// SIMATIC S7-200 project (STEP 7-Micro/WIN), CPU 224 REL 01.11

SYMBOL_TABLE USER1
ON_OFF           I0.0
X1               Q0.0
V1               Q0.1
D1               M1.0
X2               Q0.2
V2               Q0.3
D2               M1.1
END_SYMBOL_TABLE

ORGANIZATION_BLOCK MAIN:OB1
TITLE=PROGRAM COMMENTS
BEGIN
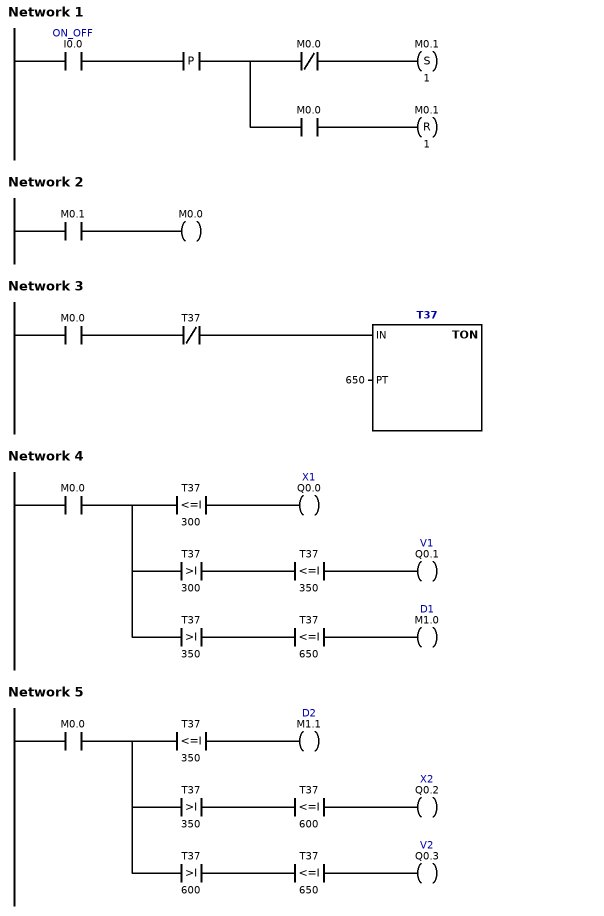
Network 1
LD     ON_OFF:I0.0
EU
LPS
AN     M0.0
S      M0.1, 1
LPP
A      M0.0
R      M0.1, 1
Network 2
LD     M0.1
=      M0.0
Network 3
LD     M0.0
AN     T37
TON    T37, 650
Network 4
LD     M0.0
LPS
AW<=   T37, 300
=      X1:Q0.0
LRD
AW>    T37, 300
AW<=   T37, 350
=      V1:Q0.1
LPP
AW>    T37, 350
AW<=   T37, 650
=      D1:M1.0
Network 5
LD     M0.0
LPS
AW<=   T37, 350
=      D2:M1.1
LRD
AW>    T37, 350
AW<=   T37, 600
=      X2:Q0.2
LPP
AW>    T37, 600
AW<=   T37, 650
=      V2:Q0.3
END_ORGANIZATION_BLOCK
